FUNCTION_BLOCK FB_Pump_RelayOnly EXTENDS FB_Pump
VAR_INPUT
END_VAR
VAR_OUTPUT
    hydrualicPump_output : ST_Pump_Output;
END_VAR
VAR
END_VAR

ACTION ExecuteState:


CASE curState OF
	eState_Idle: ExecuteState_Idle();
	eState_Startup: ExecuteState_Startup();
	eState_Running: ExecuteState_Running();
	eState_Complete: ExecuteState_Complete();
    eState_Stopping: ExecuteState_Stopping();
    eState_Stopped: ExecuteState_Stopped();
	eState_Error: ExecuteState_Error();
	eState_Independent: ExecuteState_Independent();
END_CASE
END_ACTION

ACTION ExecuteState_Complete:

END_ACTION

ACTION ExecuteState_Error:
// Set Outputs
hydrualicPump_output.On := FALSE;
END_ACTION

ACTION ExecuteState_Idle:
// Set Outputs
hydrualicPump_output.On := FALSE;
END_ACTION

ACTION ExecuteState_Independent:
// Set Outputs
hydrualicPump_output.On := FALSE;
END_ACTION

ACTION ExecuteState_Running:
// Set Outputs
hydrualicPump_output.On := TRUE;
END_ACTION

ACTION ExecuteState_Startup:

// reset timers

// set output to true
nextState := eState_Running;
END_ACTION

ACTION ExecuteState_Stopped:
nextState := eState_Idle;
END_ACTION

ACTION ExecuteState_Stopping:
nextState := eState_Stopped;
END_ACTION

METHOD getSignal : BOOL
VAR_INPUT
END_VAR
getSignal := hydrualicPump_output.On;
END_METHOD

METHOD reset : BOOL
resetAlarms();

IF curState = eState_Complete THEN
	nextState := eState_Idle;
	reset := TRUE;
ELSIF curState = eState_Error THEN
    nextState := eState_Idle;
ELSE
	reset := FALSE;
END_IF
END_METHOD

METHOD start: BOOL
VAR_INPUT
END_VAR
IF curState = eState_Idle THEN
	nextState := eState_Startup;
	start := TRUE;
ELSE
	start := FALSE;
END_IF
END_METHOD

ACTION StateTransition:
SUPER^.StateTransition();
END_ACTION

END_FUNCTION_BLOCK

(* stored: Version 1.1.0.1, ProductVersion 3.1.4024.9
   POU FB_Pump_RelayOnly: Id {bbf9f5cb-a340-456f-a981-0c6c70e04f66}, SpecialFunc None
   Folder StateMachine: Id {0f7e327f-efa4-4329-aa48-36d3216fdd27}
   Folder States: Id {9a674d99-9e31-4336-aa1e-38ca6bc25ba1}
   Action ExecuteState: Id {3291a433-6560-4362-a447-50cf99f5952a}
   Action ExecuteState_Complete: Id {785f57fe-52f1-492d-8945-58387f7b64cf}
   Action ExecuteState_Error: Id {0457ed0a-9da3-4f73-86c0-04334a7bd651}
   Action ExecuteState_Idle: Id {a81535c6-c4b3-48e7-83f0-04757990912d}
   Action ExecuteState_Independent: Id {e220d4b7-f88d-48c6-997c-7683e2fb9591}
   Action ExecuteState_Running: Id {b3869bed-62b3-4bc9-83a5-2275f062f2ef}
   Action ExecuteState_Startup: Id {44099863-9dbc-419d-9316-745ba58d4270}
   Action ExecuteState_Stopped: Id {c80c5bfd-fa3c-4da0-854d-a31eea981b5d}
   Action ExecuteState_Stopping: Id {903e1b23-df82-4512-a62b-b41f2a44bf2c}
   Method getSignal: Id {34b5af09-620e-4d91-ae26-08fbbada1ae4}
   Method reset: Id {ce3c5d84-a714-42f4-acdc-bca73ac11b2e}
   Method start: Id {93f93f60-35d6-4f62-91d6-44c0d22b6478}
   Action StateTransition: Id {75c24893-6495-4802-9ed3-914313e5eff2} *)
